// TIA Portal V18 export
// export: Created 2026-06-08T16:32:21.5263041Z, ExportSetting WithDefaults, DisplayName Totally Integrated Automation Portal, DisplayVersion V18, DisplayName TIA Portal Openness, DisplayVersion V18, DisplayName TIA Portal Version Control Interface, DisplayVersion V18, DisplayName STEP 7 Professional, DisplayVersion V18, DisplayName STEP 7 Safety, DisplayVersion V18, DisplayName WinCC Professional, DisplayVersion V18
FUNCTION_BLOCK "A_COUNTER"   // FB12, LAD
VERSION : 0.1
// stored: AutoNumber true, IsIECCheckEnabled false, UDAEnableTagReadback false
BEGIN

REGION Network 1
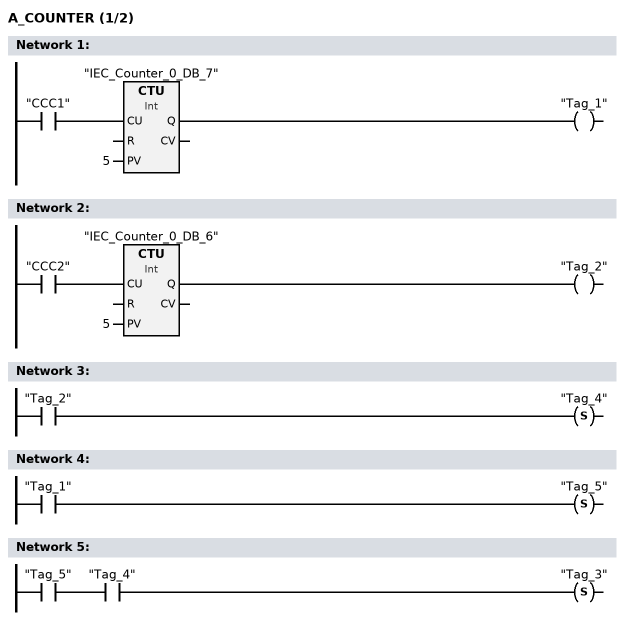
   RUNG wire#powerrail
      Contact( "CCC1" )
      { S7_Templates := "value_type := Int" } "IEC_Counter_0_DB_7".CTU(r :=, pv := 5, cv =>)
      Coil( "Tag_1" )
   END_RUNG
   // the same network as SCL:
   "IEC_Counter_0_DB_7".CTU(CU := "CCC1", PV := 5);
   "Tag_1" := "IEC_Counter_0_DB_7".Q;
END_REGION

REGION Network 2
   RUNG wire#powerrail
      Contact( "CCC2" )
      { S7_Templates := "value_type := Int" } "IEC_Counter_0_DB_6".CTU(r :=, pv := 5, cv =>)
      Coil( "Tag_2" )
   END_RUNG
   // the same network as SCL:
   "IEC_Counter_0_DB_6".CTU(CU := "CCC2", PV := 5);
   "Tag_2" := "IEC_Counter_0_DB_6".Q;
END_REGION

REGION Network 3
   RUNG wire#powerrail
      Contact( "Tag_2" )
      S_Coil( "Tag_4" )
   END_RUNG
   // the same network as SCL:
   IF "Tag_2" THEN "Tag_4" := TRUE; END_IF;
END_REGION

REGION Network 4
   RUNG wire#powerrail
      Contact( "Tag_1" )
      S_Coil( "Tag_5" )
   END_RUNG
   // the same network as SCL:
   IF "Tag_1" THEN "Tag_5" := TRUE; END_IF;
END_REGION

REGION Network 5
   RUNG wire#powerrail
      Contact( "Tag_5" )
      Contact( "Tag_4" )
      S_Coil( "Tag_3" )
   END_RUNG
   // the same network as SCL:
   IF "Tag_5" AND "Tag_4" THEN "Tag_3" := TRUE; END_IF;
END_REGION

REGION Network 6
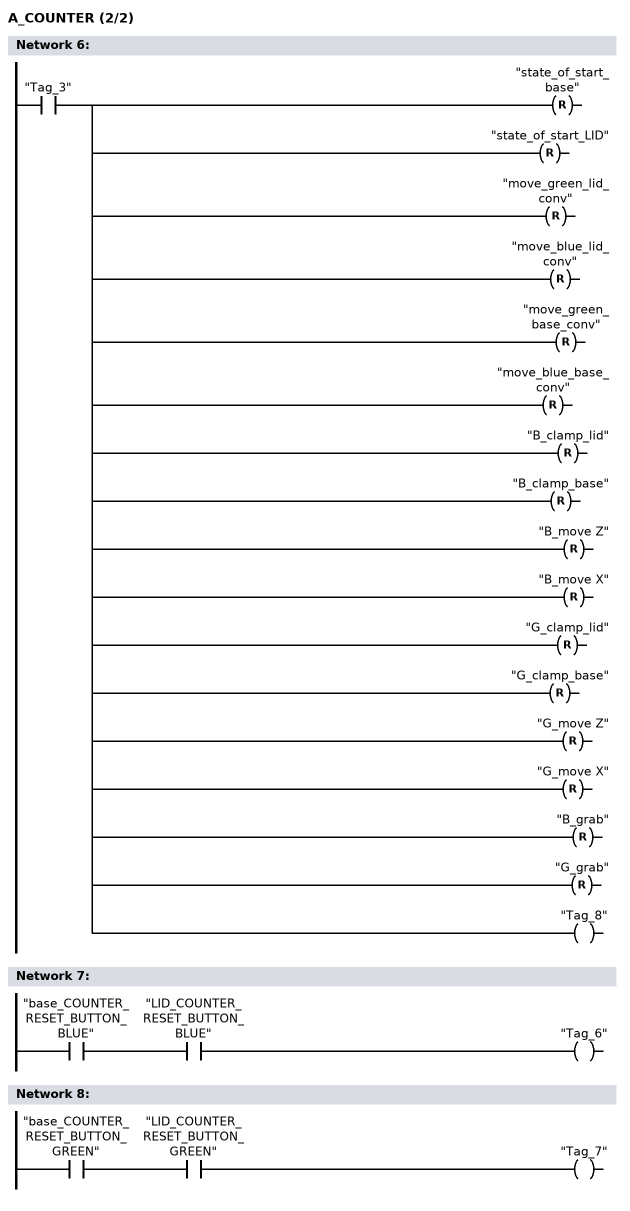
   RUNG wire#powerrail
      Contact( "Tag_3" )
      wire#w1
      R_Coil( "state_of_start_base" )
   END_RUNG
   RUNG wire#w1
      R_Coil( "state_of_start_LID" )
   END_RUNG
   RUNG wire#w1
      R_Coil( "move_green_lid_conv" )
   END_RUNG
   RUNG wire#w1
      R_Coil( "move_blue_lid_conv" )
   END_RUNG
   RUNG wire#w1
      R_Coil( "move_green_base_conv" )
   END_RUNG
   RUNG wire#w1
      R_Coil( "move_blue_base_conv" )
   END_RUNG
   RUNG wire#w1
      R_Coil( "B_clamp_lid" )
   END_RUNG
   RUNG wire#w1
      R_Coil( "B_clamp_base" )
   END_RUNG
   RUNG wire#w1
      R_Coil( "B_move Z" )
   END_RUNG
   RUNG wire#w1
      R_Coil( "B_move X" )
   END_RUNG
   RUNG wire#w1
      R_Coil( "G_clamp_lid" )
   END_RUNG
   RUNG wire#w1
      R_Coil( "G_clamp_base" )
   END_RUNG
   RUNG wire#w1
      R_Coil( "G_move Z" )
   END_RUNG
   RUNG wire#w1
      R_Coil( "G_move X" )
   END_RUNG
   RUNG wire#w1
      R_Coil( "B_grab" )
   END_RUNG
   RUNG wire#w1
      R_Coil( "G_grab" )
   END_RUNG
   RUNG wire#w1
      Coil( "Tag_8" )
   END_RUNG
   // the same network as SCL:
   IF "Tag_3" THEN
       "state_of_start_base" := FALSE;
       "state_of_start_LID" := FALSE;
       "move_green_lid_conv" := FALSE;
       "move_blue_lid_conv" := FALSE;
       "move_green_base_conv" := FALSE;
       "move_blue_base_conv" := FALSE;
       "B_clamp_lid" := FALSE;
       "B_clamp_base" := FALSE;
       "B_move Z" := FALSE;
       "B_move X" := FALSE;
       "G_clamp_lid" := FALSE;
       "G_clamp_base" := FALSE;
       "G_move Z" := FALSE;
       "G_move X" := FALSE;
       "B_grab" := FALSE;
       "G_grab" := FALSE;
   END_IF;
   "Tag_8" := "Tag_3";
END_REGION

REGION Network 7
   RUNG wire#powerrail
      Contact( "base_COUNTER_RESET_BUTTON_BLUE" )
      Contact( "LID_COUNTER_RESET_BUTTON_BLUE" )
      Coil( "Tag_6" )
   END_RUNG
   // the same network as SCL:
   "Tag_6" := "base_COUNTER_RESET_BUTTON_BLUE" AND "LID_COUNTER_RESET_BUTTON_BLUE";
END_REGION

REGION Network 8
   RUNG wire#powerrail
      Contact( "base_COUNTER_RESET_BUTTON_GREEN" )
      Contact( "LID_COUNTER_RESET_BUTTON_GREEN" )
      Coil( "Tag_7" )
   END_RUNG
   // the same network as SCL:
   "Tag_7" := "base_COUNTER_RESET_BUTTON_GREEN" AND "LID_COUNTER_RESET_BUTTON_GREEN";
END_REGION
END_FUNCTION_BLOCK
